(* Logix 5000 project; controller PLCbox vendor 1 type 14 code 149 rev 30.11; software revision 30.01; part 3 of 4 *)
(* tags used below, declared in another part *)
   Conv1Speed : REAL;
   Conv2Speed_Fast : REAL;
   Conv2Speed_Slow : REAL;
   FIO_B_IN_0 : BOOL;   // Start Button
   FIO_B_IN_1 : BOOL;   // Stop Button
   FIO_B_IN_2 : BOOL;   // System Running
   FIO_B_IN_3 : BOOL;   // Reset Button
   FIO_B_IN_4 : BOOL;
   FIO_B_OUT_0 : BOOL;   // System Running - Confirmation
   FIO_B_OUT_1 : BOOL;   // System Stopped - Confirmation
   FIO_B_OUT_2 : BOOL;   // System Faulted - Confirmation
   FIO_B_OUT_3 : BOOL;   // Send boxes
   FIO_B_OUT_4 : BOOL;
   FIO_B_OUT_5 : BOOL;
   FIO_B_OUT_6 : BOOL;
   FIO_F_OUT_0 : REAL;
   FIO_F_OUT_1 : REAL;
   IN_Loc1 : BOOL[32];
   Proj1_INT : INT[4];
   RiserBOOL : BOOL[64];
   RiserREAL : REAL[20];

PROGRAM PF525Control   (* main routine _01_Main *)
VAR
   PF525_Start_Request : BOOL;
   PowerFlex525_Start : ALIAS FOR Local:1:I.Data.0;
   PowerFlex525_Stop : ALIAS FOR Local:1:I.Data.1;
END_VAR

ROUTINE _01_Main   (* ladder *)
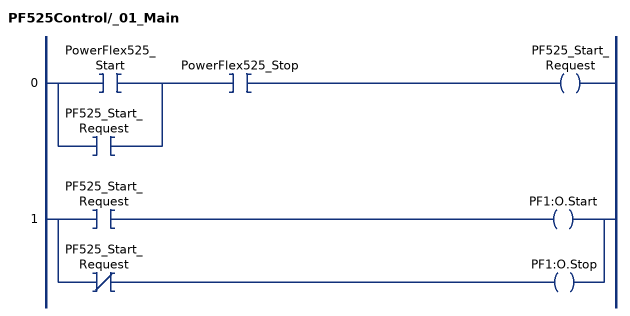
   0: [XIC(PowerFlex525_Start) ,XIC(PF525_Start_Request) ]XIC(PowerFlex525_Stop)OTE(PF525_Start_Request);
   1: [XIC(PF525_Start_Request) OTE(PF1:O.Start) ,XIO(PF525_Start_Request) OTE(PF1:O.Stop) ];
END_ROUTINE
END_PROGRAM

PROGRAM PLC_Projects   (* main routine _01_Main *)
VAR
   Proj1_TMR : TIMER[10] := ([0].PRE := 1000, [1].PRE := 1000);
END_VAR

ROUTINE _01_Main   (* ladder *)
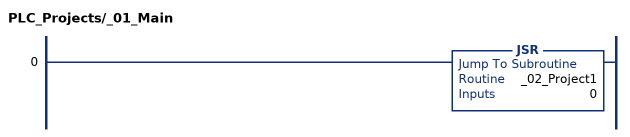
   0: JSR(_02_Project1,0);
END_ROUTINE

ROUTINE _02_Project1   (* ladder *)
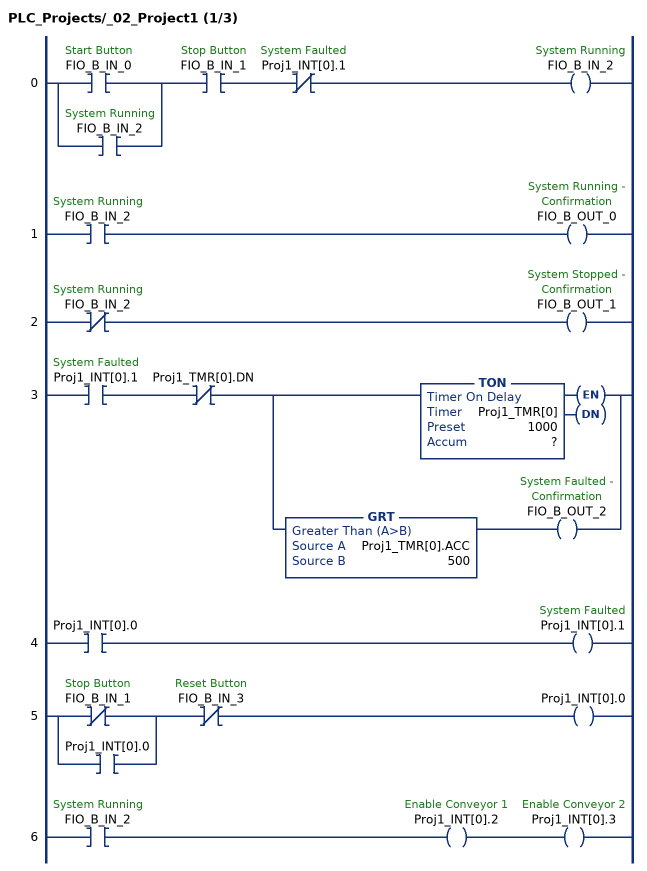
   0: [XIC(FIO_B_IN_0) ,XIC(FIO_B_IN_2) ]XIC(FIO_B_IN_1)XIO(Proj1_INT[0].1)OTE(FIO_B_IN_2);
   1: XIC(FIO_B_IN_2)OTE(FIO_B_OUT_0);
   2: XIO(FIO_B_IN_2)OTE(FIO_B_OUT_1);
   3: XIC(Proj1_INT[0].1)XIO(Proj1_TMR[0].DN)[TON(Proj1_TMR[0],?,?) ,GRT(Proj1_TMR[0].ACC,500) OTE(FIO_B_OUT_2) ];
   4: XIC(Proj1_INT[0].0)OTE(Proj1_INT[0].1);
   5: [XIO(FIO_B_IN_1) ,XIC(Proj1_INT[0].0) ]XIO(FIO_B_IN_3)OTE(Proj1_INT[0].0);
   6: XIC(FIO_B_IN_2)OTE(Proj1_INT[0].2)OTE(Proj1_INT[0].3);
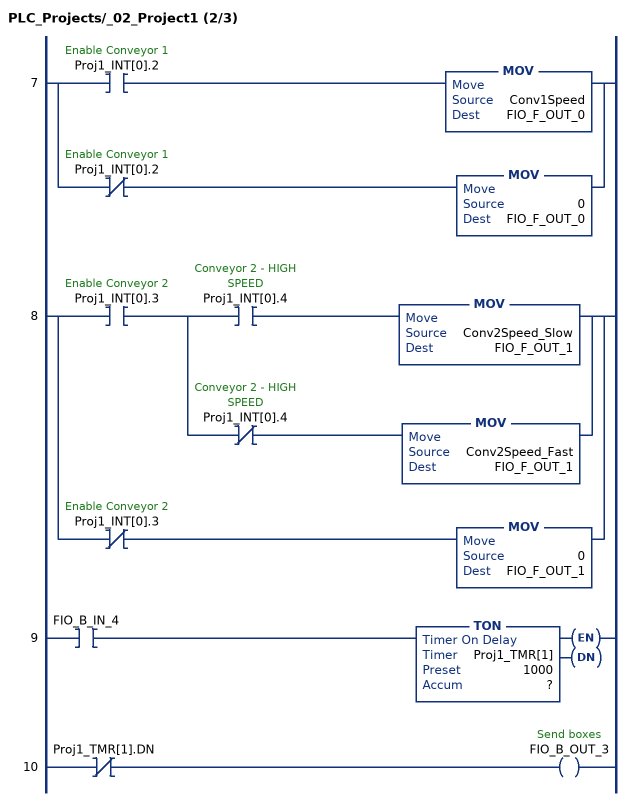
   7: [XIC(Proj1_INT[0].2) MOV(Conv1Speed,FIO_F_OUT_0) ,XIO(Proj1_INT[0].2) MOV(0,FIO_F_OUT_0) ];
   8: [XIC(Proj1_INT[0].3) [XIC(Proj1_INT[0].4) MOV(Conv2Speed_Slow,FIO_F_OUT_1) ,XIO(Proj1_INT[0].4) MOV(Conv2Speed_Fast,FIO_F_OUT_1) ] ,XIO(Proj1_INT[0].3) MOV(0,FIO_F_OUT_1) ];
   9: XIC(FIO_B_IN_4)TON(Proj1_TMR[1],?,?);
   10: XIO(Proj1_TMR[1].DN)OTE(FIO_B_OUT_3);
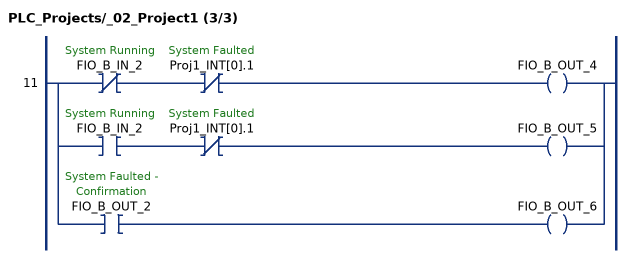
   11: [XIO(FIO_B_IN_2) XIO(Proj1_INT[0].1) OTE(FIO_B_OUT_4) ,XIC(FIO_B_IN_2) XIO(Proj1_INT[0].1) OTE(FIO_B_OUT_5) ,XIC(FIO_B_OUT_2) OTE(FIO_B_OUT_6) ];
END_ROUTINE
END_PROGRAM

PROGRAM PowerFlex525Mastery   (* main routine _01_Main *)
VAR
   Drive_Status : DINT := 2;
   Motor_Dev : REAL := 50.0;
   Motor_Fault_Timer : TIMER := (PRE := 20000);
   Motor_Faulted : BOOL := 1;
   Motor_Run : BOOL;
   Motor_SpdLim_High : REAL := 1050.0;
   Motor_SpdLim_Low : REAL := 950.0;
   Motor_Target_Speed_Fault : BOOL;
   Reset_PB : BOOL;
   Start_PB : BOOL;
   Stop_PB : BOOL;
END_VAR

ROUTINE _01_Main   (* ladder *)
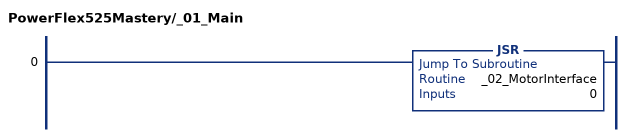
   0: JSR(_02_MotorInterface,0);
END_ROUTINE

ROUTINE _02_MotorInterface   (* ladder *)
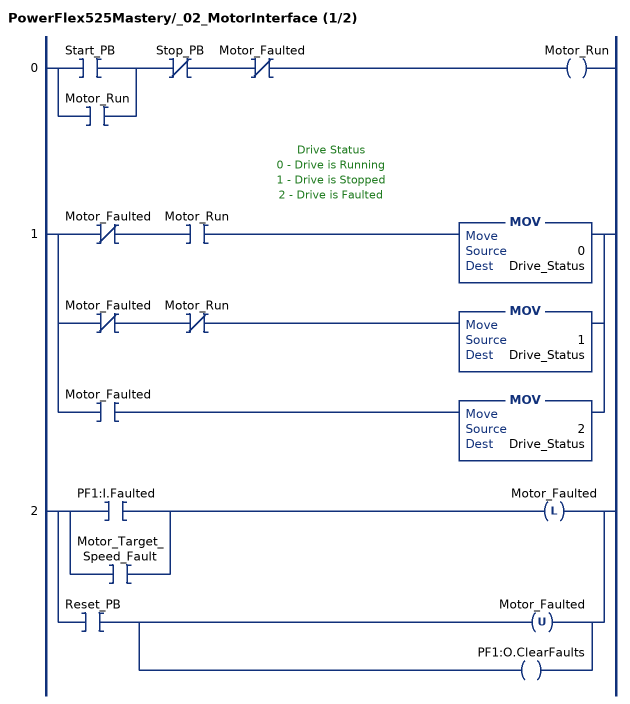
   0: [XIC(Start_PB) ,XIC(Motor_Run) ]XIO(Stop_PB)XIO(Motor_Faulted)OTE(Motor_Run);
   // Drive Status
   // 0 - Drive is Running
   // 1 - Drive is Stopped
   // 2 - Drive is Faulted
   1: [XIO(Motor_Faulted) XIC(Motor_Run) MOV(0,Drive_Status) ,XIO(Motor_Faulted) XIO(Motor_Run) MOV(1,Drive_Status) ,XIC(Motor_Faulted) MOV(2,Drive_Status) ];
   2: [[XIC(PF1:I.Faulted) ,XIC(Motor_Target_Speed_Fault) ] OTL(Motor_Faulted) ,XIC(Reset_PB) [OTU(Motor_Faulted) ,OTE(PF1:O.ClearFaults) ] ];
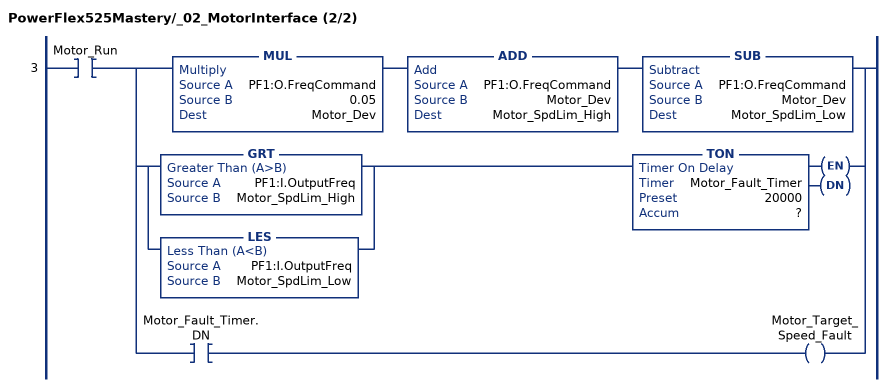
   3: XIC(Motor_Run)[MUL(PF1:O.FreqCommand,0.05,Motor_Dev) ADD(PF1:O.FreqCommand,Motor_Dev,Motor_SpdLim_High) SUB(PF1:O.FreqCommand,Motor_Dev,Motor_SpdLim_Low) ,[GRT(PF1:I.OutputFreq,Motor_SpdLim_High) ,LES(PF1:I.OutputFreq,Motor_SpdLim_Low) ] TON(Motor_Fault_Timer,?,?) ,XIC(Motor_Fault_Timer.DN) OTE(Motor_Target_Speed_Fault) ];
END_ROUTINE
END_PROGRAM

PROGRAM Riser   (* main routine _01_Main *)

ROUTINE _01_Main   (* ladder *)
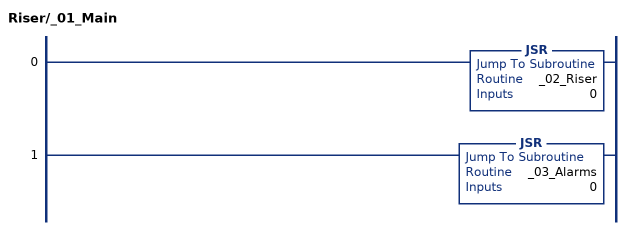
   0: JSR(_02_Riser,0);
   1: JSR(_03_Alarms,0);
END_ROUTINE

ROUTINE _02_Riser   (* ladder *)
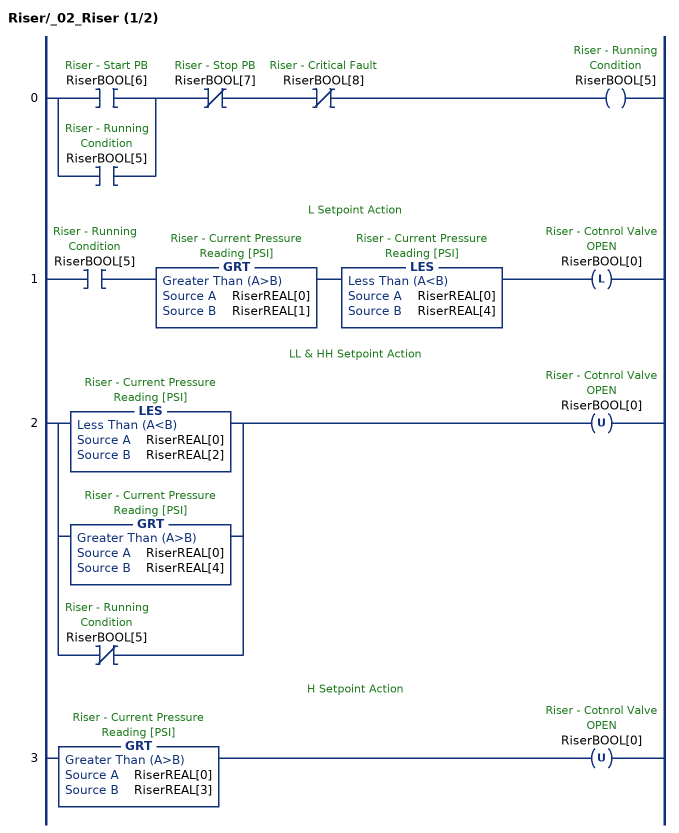
   0: [XIC(RiserBOOL[6]) ,XIC(RiserBOOL[5]) ]XIO(RiserBOOL[7])XIO(RiserBOOL[8])OTE(RiserBOOL[5]);
   // L Setpoint Action
   1: XIC(RiserBOOL[5])GRT(RiserREAL[0],RiserREAL[1])LES(RiserREAL[0],RiserREAL[4])OTL(RiserBOOL[0]);
   // LL & HH Setpoint Action
   2: [LES(RiserREAL[0],RiserREAL[2]) ,GRT(RiserREAL[0],RiserREAL[4]) ,XIO(RiserBOOL[5]) ]OTU(RiserBOOL[0]);
   // H Setpoint Action
   3: GRT(RiserREAL[0],RiserREAL[3])OTU(RiserBOOL[0]);
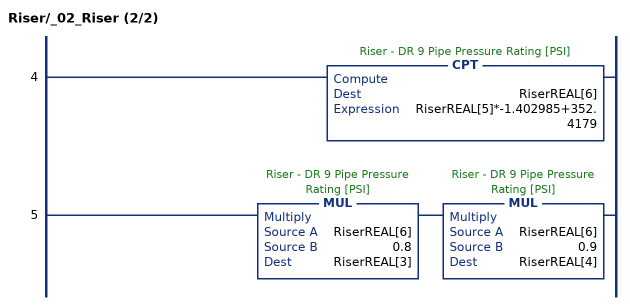
   4: CPT(RiserREAL[6],RiserREAL[5]*-1.402985+352.4179);
   5: MUL(RiserREAL[6],0.8,RiserREAL[3])MUL(RiserREAL[6],0.9,RiserREAL[4]);
END_ROUTINE

ROUTINE _03_Alarms   (* ladder *)
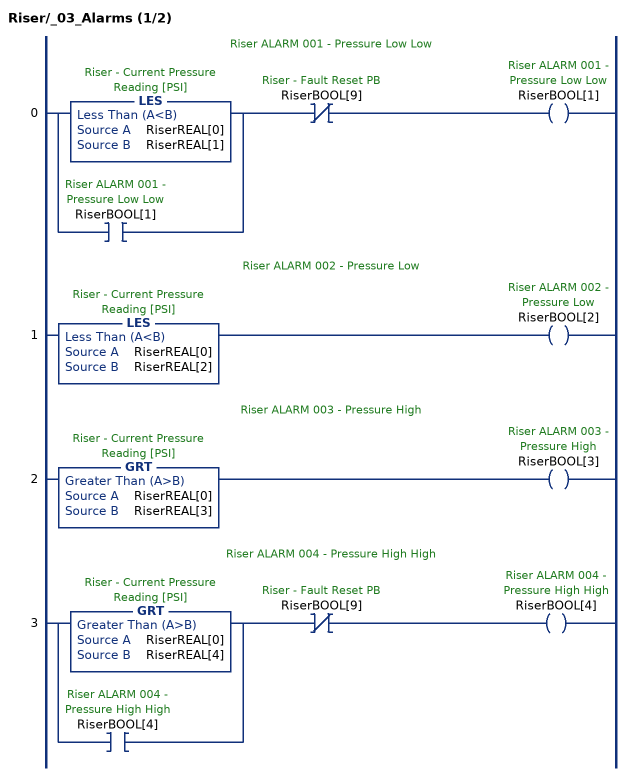
   // Riser ALARM 001 - Pressure Low Low
   0: [LES(RiserREAL[0],RiserREAL[1]) ,XIC(RiserBOOL[1]) ]XIO(RiserBOOL[9])OTE(RiserBOOL[1]);
   // Riser ALARM 002 - Pressure Low
   1: LES(RiserREAL[0],RiserREAL[2])OTE(RiserBOOL[2]);
   // Riser ALARM 003 - Pressure High
   2: GRT(RiserREAL[0],RiserREAL[3])OTE(RiserBOOL[3]);
   // Riser ALARM 004 - Pressure High High
   3: [GRT(RiserREAL[0],RiserREAL[4]) ,XIC(RiserBOOL[4]) ]XIO(RiserBOOL[9])OTE(RiserBOOL[4]);
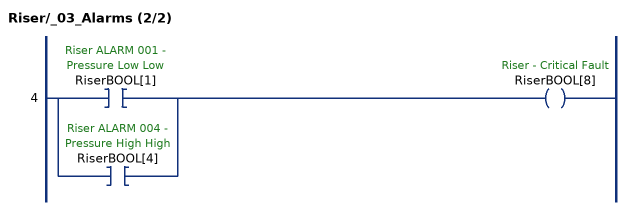
   4: [XIC(RiserBOOL[1]) ,XIC(RiserBOOL[4]) ]OTE(RiserBOOL[8]);
END_ROUTINE
END_PROGRAM

PROGRAM RPiEdgeIgnition   (* main routine _01_Main *)
VAR
   RPiEdge_BOOL : BOOL[256] := ([0] := 1);
   RPiEdge_BOOL2 : BOOL[256] := ([0] := 1, [1] := 1, [2] := 1, [3] := 1, [5] := 1, [9] := 1, [14] := 1, [21] := 1, [23] := 1);
   RPiEdge_DINT : DINT[50] := ([0] := 3);
   RPiEdge_REAL : REAL[50] := ([0] := 1231.0, [2] := 34535.457, [4] := 35345.45, [7] := 3213.63);
   RPiEdge_STRING : STRING[20] := ([0] := 'Raw Materials Station 1', [1] := 'Raw Materials Station 2', [2] := 'Raw Materials Station 3', [3] := 'Filler', [4] := 'Wrapper', [5] := 'Barcode Verification', [6] := 'Sealer', [7] := 'Quality Reject Station', [8] := 'Case Packer', [9] := 'Palletizer', [10] := 'Spare 1', [11] := 'Spare 2');
   RPiS_BOOL : BOOL[256];
        [1]   // System 1 - Stop
        [0]   // System 1 - Start
        [6]   // System 1 - Fault
        [4]   // System 1 - Auto Run Permissive
        [2]   // System 1 - Enabled
        [3]   // System 1 - Manual
        [5]   // System 1 - Faulted
        [7]   // System 1 - Fault Reset
END_VAR

ROUTINE _01_Main   (* ladder *)
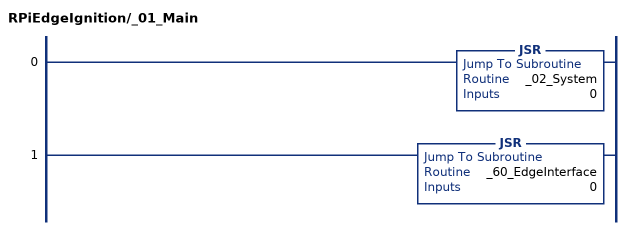
   0: JSR(_02_System,0);
   1: JSR(_60_EdgeInterface,0);
END_ROUTINE

ROUTINE _02_System   (* ladder *)
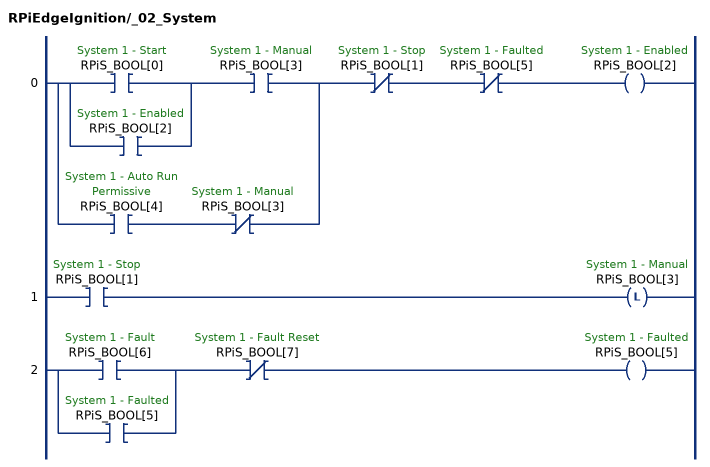
   0: [[XIC(RPiS_BOOL[0]) ,XIC(RPiS_BOOL[2]) ] XIC(RPiS_BOOL[3]) ,XIC(RPiS_BOOL[4]) XIO(RPiS_BOOL[3]) ]XIO(RPiS_BOOL[1])XIO(RPiS_BOOL[5])OTE(RPiS_BOOL[2]);
   1: XIC(RPiS_BOOL[1])OTL(RPiS_BOOL[3]);
   2: [XIC(RPiS_BOOL[6]) ,XIC(RPiS_BOOL[5]) ]XIO(RPiS_BOOL[7])OTE(RPiS_BOOL[5]);
END_ROUTINE

ROUTINE _30_Faults   (* ladder *)
END_ROUTINE

ROUTINE _60_EdgeInterface   (* ladder *)
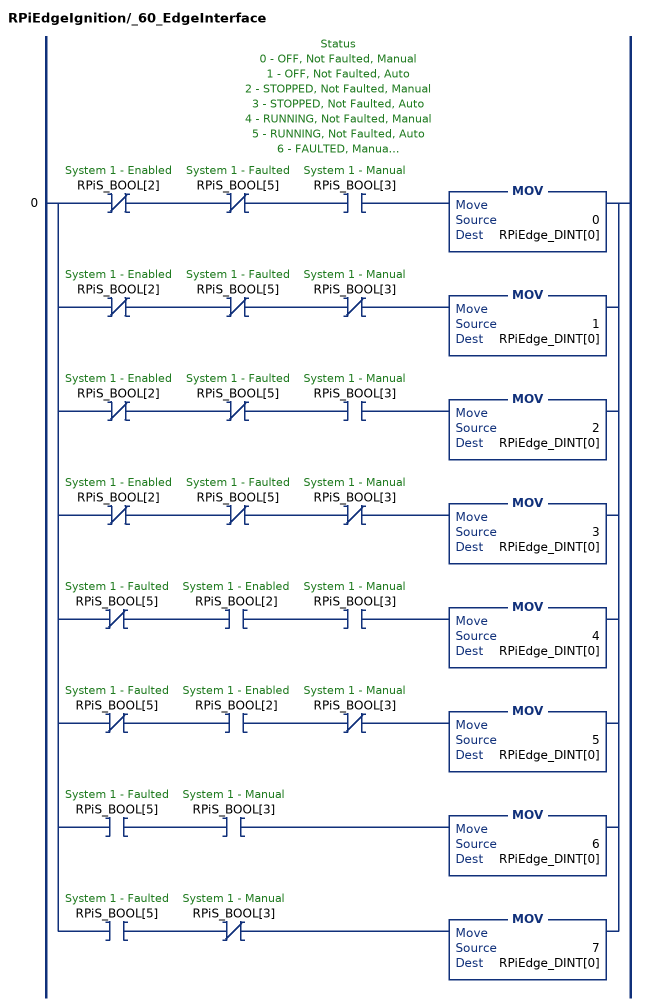
   // Status
   // 0 - OFF, Not Faulted, Manual
   // 1 - OFF, Not Faulted, Auto
   // 2 - STOPPED, Not Faulted, Manual
   // 3 - STOPPED, Not Faulted, Auto
   // 4 - RUNNING, Not Faulted, Manual
   // 5 - RUNNING, Not Faulted, Auto
   // 6 - FAULTED, Manual
   // 7 - FAULTED, Auto
   0: [XIO(RPiS_BOOL[2]) XIO(RPiS_BOOL[5]) XIC(RPiS_BOOL[3]) MOV(0,RPiEdge_DINT[0]) ,XIO(RPiS_BOOL[2]) XIO(RPiS_BOOL[5]) XIO(RPiS_BOOL[3]) MOV(1,RPiEdge_DINT[0]) ,XIO(RPiS_BOOL[2]) XIO(RPiS_BOOL[5]) XIC(RPiS_BOOL[3]) MOV(2,RPiEdge_DINT[0]) ,XIO(RPiS_BOOL[2]) XIO(RPiS_BOOL[5]) XIO(RPiS_BOOL[3]) MOV(3,RPiEdge_DINT[0]) ,XIO(RPiS_BOOL[5]) XIC(RPiS_BOOL[2]) XIC(RPiS_BOOL[3]) MOV(4,RPiEdge_DINT[0]) ,XIO(RPiS_BOOL[5]) XIC(RPiS_BOOL[2]) XIO(RPiS_BOOL[3]) MOV(5,RPiEdge_DINT[0]) ,XIC(RPiS_BOOL[5]) XIC(RPiS_BOOL[3]) MOV(6,RPiEdge_DINT[0]) ,XIC(RPiS_BOOL[5]) XIO(RPiS_BOOL[3]) MOV(7,RPiEdge_DINT[0]) ];
END_ROUTINE
END_PROGRAM

PROGRAM ST_Practice   (* main routine _01_Main *)
VAR
   AScaled : REAL := 93.75;
   BOOL : BOOL[64];
   LocalBOOL : BOOL[64] := ([6] := 1);
   LocalDINT : DINT[20] := ([0] := 95);
   LocDINT : DINT[20] := ([0] := 5, [2] := -4, [4] := 15, [5] := 5, [6] := 125, [7] := 1, [8] := 58);
   LocOut : DINT[20];
   LogicDINT : DINT[100];
   MotorRUN : DINT;
   MotorRUN2 : BOOL := 1;
   MRT_Stop : BOOL;
   MTR1 : BOOL[64];
        [1]   // Motor - Stop PB
        [0]   // Motor - Start PB
        [2]   // Motor - Running
   MTR_Run : BOOL;
   MTR_Start : BOOL;
   NewTagBOOL : BOOL;
   NewTagBOOL2 : BOOL;
   NewTagDINT : DINT := 1242;
   NewTagINT : IMC := (PVEUMax := 100.0, SPHLimit := 100.0, RatioProg := 1.0, RatioOper := 1.0, RatioHLimit := 1.0, RatioLLimit := 1.0, CVEUMax := 100.0, CVHLimit := 100.0, ModelGain := 1.0, RTSTime := 1, AtuneTimeLimit := 60.0, NoiseLevel := 1, CVStepSize := 10.0, ResponseSpeed := 1, Factor := 100.0);
   NewTagSTRING : STRING := 'A';
   NewTagSTRING2 : STRING;
   NewTagVar : DINT := 44;
   Running : BOOL;
   StartPB : BOOL;
   StopButton : BOOL;
   StopPB : DINT;
   StopPB2 : BOOL;
   TagBOOL : BOOL := 1;
   TagBOOL2 : BOOL := 1;
   TagDINT : DINT := 34;
   TagINT : INT := 34;
   TagINT2 : INT := 56;
   TagSTRING : STRING;
   TempC : REAL := 22.222221;
   TempF : REAL := 72.0;
END_VAR

ROUTINE _01_Main   (* ladder *)
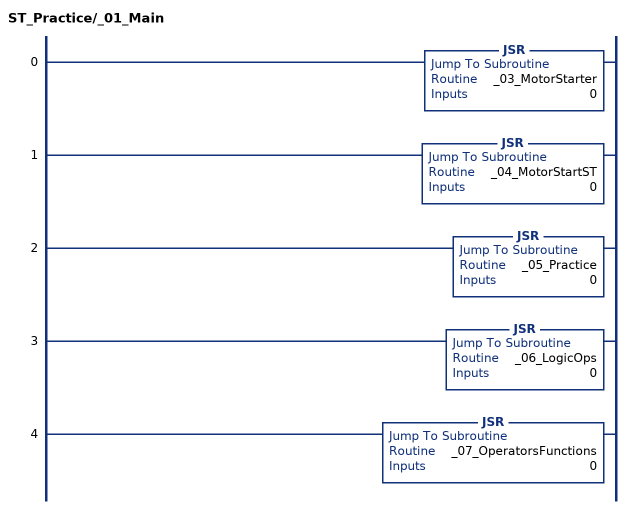
   0: JSR(_03_MotorStarter,0);
   1: JSR(_04_MotorStartST,0);
   2: JSR(_05_Practice,0);
   3: JSR(_06_LogicOps,0);
   4: JSR(_07_OperatorsFunctions,0);
END_ROUTINE

ROUTINE _02_InputDef   (* structured text *)
   IN_Loc1[0] := Local:1:I.Data.0; //Start PB
   IN_Loc1[1] := Local:1:I.Data.1; //Stop PB
   IN_Loc1[2] := Local:1:I.Data.2; //Reset from HMI
   IN_Loc1[3] := Local:1:I.Data.3; //
   IN_Loc1[4] := Local:1:I.Data.4; //
   IN_Loc1[5] := Local:1:I.Data.5; //
   IN_Loc1[6] := Local:1:I.Data.6; //
   IN_Loc1[7] := Local:1:I.Data.7; //
   IN_Loc1[8] := Local:1:I.Data.8; //
   IN_Loc1[9] := Local:1:I.Data.9; //
   IN_Loc1[10] := Local:1:I.Data.10; //
   IN_Loc1[11] := Local:1:I.Data.11; //
   IN_Loc1[12] := Local:1:I.Data.12; //
   IN_Loc1[13] := Local:1:I.Data.13; //
   IN_Loc1[14] := Local:1:I.Data.14; //
   IN_Loc1[15] := Local:1:I.Data.15; //
END_ROUTINE

ROUTINE _03_MotorStarter   (* ladder *)
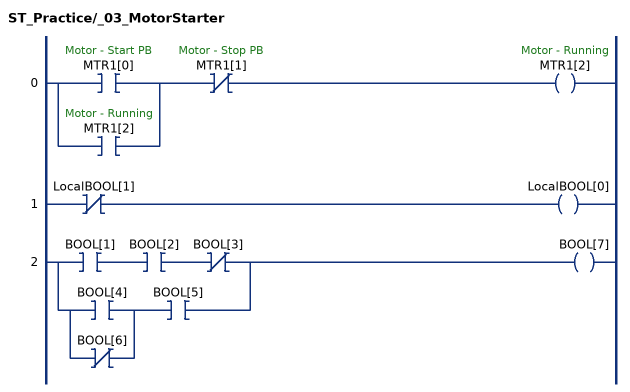
   0: [XIC(MTR1[0]) ,XIC(MTR1[2]) ]XIO(MTR1[1])OTE(MTR1[2]);
   1: XIO(LocalBOOL[1])OTE(LocalBOOL[0]);
   2: [XIC(BOOL[1]) XIC(BOOL[2]) XIO(BOOL[3]) ,[XIC(BOOL[4]) ,XIO(BOOL[6]) ] XIC(BOOL[5]) ]OTE(BOOL[7]);
END_ROUTINE
